{attribute 'pack_mode' := '2'}
TYPE PackTwo :
STRUCT
	b1  : BOOL;
	d1  : DWORD;
	b2  : BOOL;
	lw1 : LWORD;
END_STRUCT
END_TYPE

(* stored: Version 1.1.0.1, ProductVersion 3.1.4024.13
   DUT PackTwo: Id {a1b2c3d4-0000-4000-8000-000000000002} *)
